SYSTEM SERVER_HMI_NEW (* System Configuration *)
  (* Standard: 61499-1 *)
  (* Version 0.3, 2003-12-05, JHC, Rockwell Automation, Renamed from NEWSYSTEM. *)
  (* Version 0.2, 2002-11-05, JHC, Rockwell Automation, Fixed missing (empty) FBD in Application. *)
  (* Version 0.1, 2002-01-17, JHC, Rockwell Automation, Minor cleanup *)
  (* Version 0.0, 2000-05-27, JHC, Rockwell Automation *)
  APPLICATION APP1
  END_APPLICATION
  DEVICE WORKER_HMI_DEVICE : FRAME_DEVICE(BOUNDS := [1100,300,600,400], GRID := [1,1])
    RESOURCE WORKER_HMI_PROCESSOR : PANEL_RESOURCE(ROWS := 6, COLS := 2)
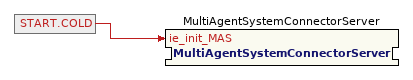
      FBS
        MultiAgentSystemConnectorServer : MultiAgentSystemConnectorServer;
      END_FBS
      EVENT_CONNECTIONS
        START.COLD TO MultiAgentSystemConnectorServer.ie_init_MAS;
      END_CONNECTIONS
    END_RESOURCE
  END_DEVICE
END_SYSTEM
